FUNCTION_BLOCK FB_Robot
VAR_INPUT
	bEnable: BOOL;
	bReset: BOOL;
END_VAR
VAR_OUTPUT
	bBusy: BOOL;
	bError: BOOL;
END_VAR
VAR
	fb_Wheel_1: FB_Wheel;
	fb_Wheel_2: FB_Wheel;
	fb_Wheel_3: FB_Wheel;
	fb_Wheel_4: FB_Wheel;
END_VAR

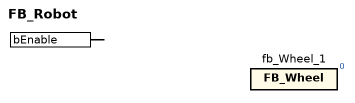
fb_Wheel_1(); // FB_Wheel
// bEnable: input not connected

END_FUNCTION_BLOCK

(* stored: Version 1.1.0.1, ProductVersion 3.1.4024.11
   POU FB_Robot: Id {8cab247d-fbc9-49dc-a66b-b822d742e76a}, SpecialFunc None *)
